{attribute 'GeneratedUsingTerminal: BK1120-0000-0001'}
{attribute addProperty BoxType "BK1120-0000-0001"}
{attribute addProperty Id "Term_375_KL1002KL1002_BB38DA8F0"}
{attribute addProperty CRC "1995569387"}
{attribute addProperty Size "0"}
TYPE A_0002_BK1120_0000_0001_76F1F8EB EXTENDS BK1120_A2FCADE7 :
STRUCT
	{attribute addProperty Name "Term_375_KL1002"}
	Term_375_KL1002 : KL1002_BB38DA8F;
END_STRUCT
END_TYPE

(* stored: Version 1.2.0.0, ProductVersion 3.1.4024.9
   DUT A_0002_BK1120_0000_0001_76F1F8EB: Id {9c9143e3-606a-44c1-8e7b-ccda521d2efb} *)
